TYPE ST_Settings :
STRUCT
	//Timeout settings
	tCameraTimeout			:TIME;
	tConveyorTimeout		:TIME;
	tPickClampTimeout		:TIME;
	tPlaceClampTimeout		:TIME;
	tFeederTimeout			:TIME;
	tRobotTimeout			:TIME;
	
	//Process settings
	tGreasingPulseTime		:TIME;
END_STRUCT
END_TYPE

(* stored: Version 1.1.0.1
   DUT ST_Settings: Id {9470d0d5-a718-40c4-9002-671168cc1c45} *)
